// TIA Portal project "ElevatorSimulatorBir" (V17)
// Vorlageprojekt für das Buch mit Zielsystem S7-1200

(* hardware
DEVICE "S7-1200-Station_1"  S7-1200 Station
   slot 0: "Baugruppenträger_0"  Rack  V1.0
   slot 1: "PLC_1"  CPU 1211C DC/DC/DC  6ES7 211-1AE40-0XB0  V4.1
*)

// ===== PLC "PLC_1"  CPU 1211C DC/DC/DC =====

VAR_GLOBAL   // PLC tag table "Standard-Variablentabelle"
   "ROLL CONVEYOR 1" AT %A0.0 : Bool;
   "STOP BUTTON 1" AT %E0.0 : Bool;
   "START BUTTON 1" AT %E0.1 : Bool;
   "Tag_4" AT %M0.0 : Bool;
   "Tag_1" AT %M0.1 : Bool;
   "ELEVATOR 1 (RIGHT LIMIT)" AT %I0.2 : Bool;
   "ELEVATOR 1 (LEFT LIMIT)" AT %I0.3 : Bool;
   "ELEVATOR 1 (-)" AT %Q0.1 : Bool;
   "KAT SENSÖRLERİ" AT %IB2 : Byte;
   "Tag_3" AT %M10.0 : Bool;
   "Tag_5" AT %M18.0 : Bool;
   "Tag_6" AT %M10.2 : Bool;
   "Tag_2" AT %MB15 : Byte;
   "ELEVATOR 1 (UP)" AT %Q0.2 : Bool;
   "ELEVATOR 1 (DOWN)" AT %Q0.3 : Bool;
   "CAGIRMA BUTONU KAT 2" AT %I3.1 : Bool;
   "Tag_8" AT %M36.0 : Bool;
   "Tag_9" AT %M36.1 : Bool;
   "CAGIRMA BUTONU KAT 3" AT %I3.2 : Bool;
   "Tag_11" AT %M36.2 : Bool;
   "CAGIRMA BUTONU KAT 4" AT %I3.3 : Bool;
   "Tag_7" AT %M10.5 : Bool;
END_VAR

FUNCTION "MHJ-PLC-Lab-Function-S71200" : Void   // FC9000, SCL
{ S7_Optimized_Access := 'TRUE' }
VERSION : 0.1
   VAR_TEMP
      rdTimeReturn : Int;
      outputTime : DTL;
      SyncVal : Byte;
      forVal : Int;
      forVal_2 : Int;
      Value : Byte;
   END_VAR
   VAR CONSTANT
      CompVal : Byte := 16#34;
      Value_01 : Byte := 16#11;
      Value_01_DW : DWord := 16#A165_D992;
      Value_02_DW : DWord := 16#58BE_4401;
   END_VAR
BEGIN

   #Value:=PEEK(area := 16#82,
        dbNumber := 0,
        byteOffset := 511);
   #Value := #Value + 1;

   POKE(area := 16#82,
        dbNumber := 0,
        byteOffset := 511,
        value := #Value);

   POKE(area:=16#81,
        dbNumber:=0,
        byteOffset:=1016,
        value:=#Value_01_DW);
   POKE(area := 16#81,
        dbNumber := 0,
        byteOffset := 1020,
        value := #Value_02_DW);

   POKE(area := 16#81,
        dbNumber := 0,
        byteOffset := 511,
        value := B#16#00);

   FOR #forVal := 0 TO 120 DO
       FOR #forVal_2:=0 TO 10 DO
           #rdTimeReturn:=RD_SYS_T(#outputTime);
           #rdTimeReturn := WR_SYS_T(#outputTime);
           #rdTimeReturn := RD_SYS_T(#outputTime);
           #rdTimeReturn := WR_SYS_T(#outputTime);
       END_FOR;
       #SyncVal:= PEEK(area := 16#81,
                      dbNumber := 0,
                      byteOffset := 511);
       IF #SyncVal = #CompVal THEN
          GOTO M_1;
       END_IF;
   END_FOR;
   RETURN;

   M_1:
   POKE(area := 16#81,
        dbNumber := 0,
        byteOffset := 511,
        value := B#16#0);
END_FUNCTION

ORGANIZATION_BLOCK "Main"   // OB1, LAD, ProgramCycle
TITLE = "Main Program Sweep (Cycle)"
{ S7_Optimized_Access := 'TRUE' }
VERSION : 0.1
   VAR_INPUT
      Initial_Call : Bool;   // Initial call of this OB
      Remanence : Bool;   // =True, if remanent data are available
   END_VAR
   VAR_TEMP   // added for the SCL form of the ladder/FBD networks
      _w1 : Bool;
   END_VAR
BEGIN

REGION Network 1: Konnektierungsbaustein für PLC-Lab
   // Im Netzwerk 1 wird der Konnektierungsbaustein für PLC-Lab aufgerufen.
   // Dieser Aufruf darf nicht entfernt werden!
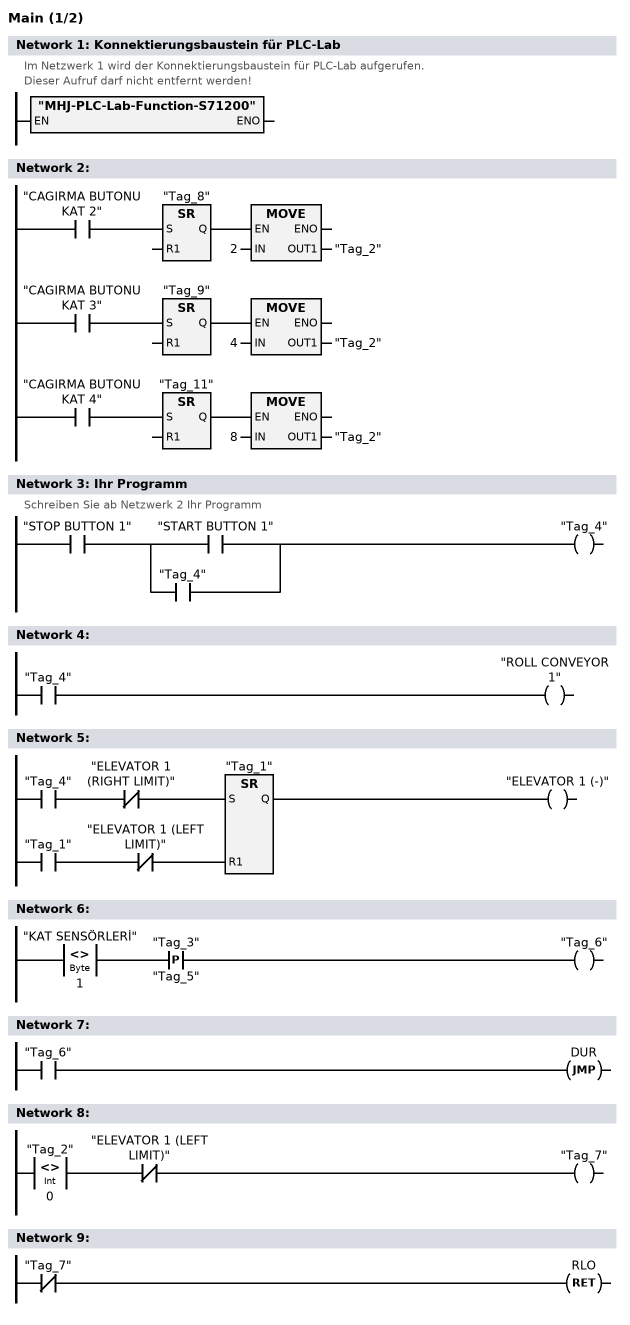
   RUNG wire#powerrail
      "MHJ-PLC-Lab-Function-S71200"()
   END_RUNG
   // the same network as SCL:
   "MHJ-PLC-Lab-Function-S71200"();
END_REGION

REGION Network 2
   RUNG wire#powerrail
      Contact( "CAGIRMA BUTONU KAT 2" )
      S_SR(operand := "Tag_8", r1 :=)
      Move(in := 2, out1 => "Tag_2")
   END_RUNG
   RUNG wire#powerrail
      Contact( "CAGIRMA BUTONU KAT 3" )
      S_SR(operand := "Tag_9", r1 :=)
      Move(in := 4, out1 => "Tag_2")
   END_RUNG
   RUNG wire#powerrail
      Contact( "CAGIRMA BUTONU KAT 4" )
      S_SR(operand := "Tag_11", r1 :=)
      Move(in := 8, out1 => "Tag_2")
   END_RUNG
   // the same network as SCL:
   IF "CAGIRMA BUTONU KAT 2" THEN
       "Tag_8" := TRUE;   // SR flip-flop
   END_IF;
   IF "Tag_8" THEN "Tag_2" := 2; END_IF;
   IF "CAGIRMA BUTONU KAT 3" THEN
       "Tag_9" := TRUE;   // SR flip-flop
   END_IF;
   IF "Tag_9" THEN "Tag_2" := 4; END_IF;
   IF "CAGIRMA BUTONU KAT 4" THEN
       "Tag_11" := TRUE;   // SR flip-flop
   END_IF;
   IF "Tag_11" THEN "Tag_2" := 8; END_IF;
END_REGION

REGION Network 3: Ihr Programm
   // Schreiben Sie ab Netzwerk 2 Ihr Programm
   RUNG wire#powerrail
      Contact( "STOP BUTTON 1" )
      wire#w1
      Contact( "START BUTTON 1" )
      wire#w2
      Coil( "Tag_4" )
   END_RUNG
   RUNG wire#w1
      Contact( "Tag_4" )
   END_RUNG wire#w2
   // the same network as SCL:
   "Tag_4" := "STOP BUTTON 1" AND ("START BUTTON 1" OR "Tag_4");
END_REGION

REGION Network 4
   RUNG wire#powerrail
      Contact( "Tag_4" )
      Coil( "ROLL CONVEYOR 1" )
   END_RUNG
   // the same network as SCL:
   "ROLL CONVEYOR 1" := "Tag_4";
END_REGION

REGION Network 5
   RUNG wire#powerrail
      Contact( "Tag_4" )
      I_Contact( "ELEVATOR 1 (RIGHT LIMIT)" )
      S_SR(operand := "Tag_1", r1 := wire#w1)
      Coil( "ELEVATOR 1 (-)" )
   END_RUNG
   RUNG wire#powerrail
      Contact( "Tag_1" )
      I_Contact( "ELEVATOR 1 (LEFT LIMIT)" )
   END_RUNG wire#w1
   // the same network as SCL:
   #_w1 := "Tag_1" AND NOT "ELEVATOR 1 (LEFT LIMIT)";
   IF "Tag_4" AND NOT "ELEVATOR 1 (RIGHT LIMIT)" THEN
       "Tag_1" := TRUE;   // SR flip-flop
   END_IF;
   IF #_w1 THEN "Tag_1" := FALSE; END_IF;
   "ELEVATOR 1 (-)" := "Tag_1";
END_REGION

REGION Network 6
   RUNG wire#powerrail
      { S7_Templates := "SrcType := Byte" } NE_Contact(in1 := "KAT SENSÖRLERİ", in2 := 1)
      P_Contact(operand := "Tag_3", bit := "Tag_5")
      Coil( "Tag_6" )
   END_RUNG
   // the same network as SCL:
   #_w1 := ("KAT SENSÖRLERİ" <> 1) AND "Tag_3" AND NOT "Tag_5";   // rising edge of "Tag_3"
   "Tag_5" := "Tag_3";
   "Tag_6" := #_w1;
END_REGION

REGION Network 7
   RUNG wire#powerrail
      Contact( "Tag_6" )
      JumpCoil( DUR )
   END_RUNG
   // the same network as SCL:
   IF "Tag_6" THEN GOTO DUR; END_IF;
END_REGION

REGION Network 8
   RUNG wire#powerrail
      { S7_Templates := "SrcType := Int" } NE_Contact(in1 := "Tag_2", in2 := 0)
      I_Contact( "ELEVATOR 1 (LEFT LIMIT)" )
      Coil( "Tag_7" )
   END_RUNG
   // the same network as SCL:
   "Tag_7" := ("Tag_2" <> 0) AND NOT "ELEVATOR 1 (LEFT LIMIT)";
END_REGION

REGION Network 9
   IF NOT "Tag_7" THEN
       ENO := TRUE;
       RETURN;
   END_IF;
END_REGION

REGION Network 10
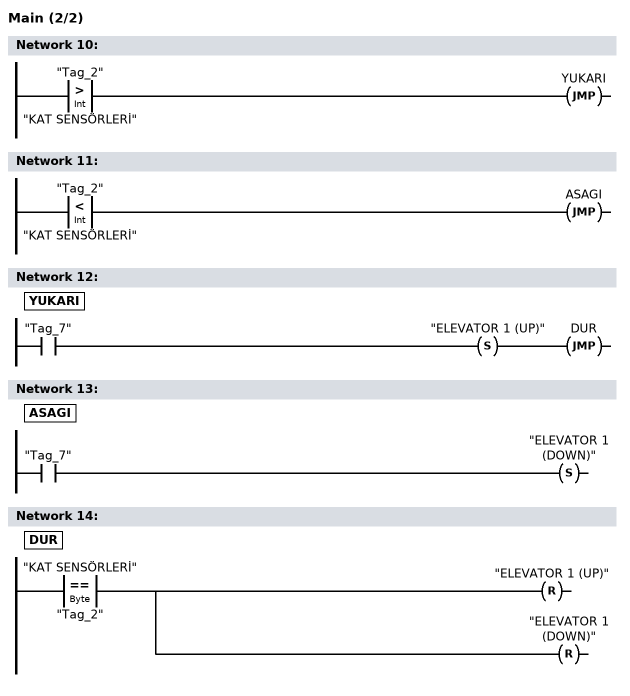
   RUNG wire#powerrail
      { S7_Templates := "SrcType := Int" } GT_Contact(in1 := "Tag_2", in2 := "KAT SENSÖRLERİ")
      JumpCoil( YUKARI )
   END_RUNG
   // the same network as SCL:
   IF "Tag_2" > "KAT SENSÖRLERİ" THEN GOTO YUKARI; END_IF;
END_REGION

REGION Network 11
   RUNG wire#powerrail
      { S7_Templates := "SrcType := Int" } LT_Contact(in1 := "Tag_2", in2 := "KAT SENSÖRLERİ")
      JumpCoil( ASAGI )
   END_RUNG
   // the same network as SCL:
   IF "Tag_2" < "KAT SENSÖRLERİ" THEN GOTO ASAGI; END_IF;
END_REGION

REGION Network 12
   Label( YUKARI )
   RUNG wire#powerrail
      Contact( "Tag_7" )
      S_Coil( "ELEVATOR 1 (UP)" )
      JumpCoil( DUR )
   END_RUNG
   // the same network as SCL:
   YUKARI:
   IF "Tag_7" THEN
       "ELEVATOR 1 (UP)" := TRUE;
       GOTO DUR;
   END_IF;
END_REGION

REGION Network 13
   Label( ASAGI )
   RUNG wire#powerrail
      Contact( "Tag_7" )
      S_Coil( "ELEVATOR 1 (DOWN)" )
   END_RUNG
   // the same network as SCL:
   ASAGI:
   IF "Tag_7" THEN "ELEVATOR 1 (DOWN)" := TRUE; END_IF;
END_REGION

REGION Network 14
   Label( DUR )
   RUNG wire#powerrail
      { S7_Templates := "SrcType := Byte" } EQ_Contact(in1 := "KAT SENSÖRLERİ", in2 := "Tag_2")
      wire#w1
      R_Coil( "ELEVATOR 1 (UP)" )
   END_RUNG
   RUNG wire#w1
      R_Coil( "ELEVATOR 1 (DOWN)" )
   END_RUNG
   // the same network as SCL:
   DUR:
   IF "KAT SENSÖRLERİ" = "Tag_2" THEN
       "ELEVATOR 1 (UP)" := FALSE;
       "ELEVATOR 1 (DOWN)" := FALSE;
   END_IF;
END_REGION
END_ORGANIZATION_BLOCK